// TIA Portal V15.1 export
// export: Created 2026-01-15T16:29:47.7440126Z, ExportSetting WithDefaults, WithReadOnly, DisplayName Totally Integrated Automation Portal, DisplayVersion V15.1 Update 8, DisplayName TIA Portal Openness, DisplayVersion V15.1 Update 8, DisplayName STEP 7 Professional, DisplayVersion V15.1 Update 8, DisplayName WinCC Advanced, DisplayVersion V15.1 Update 8
FUNCTION "FCXL_CCD_FD1" : Void   // FC10, LAD
{ S7_Optimized_Access := 'TRUE' }
VERSION : 0.1
// stored: AutoNumber true, CodeModifiedDate 2026-01-15T16:25:54.9008625Z, CompileDate 2026-01-15T16:25:54.9411388Z, CreationDate 2026-01-15T16:24:02.4619467Z, HandleErrorsWithinBlock false, InterfaceModifiedDate 2024-08-08T03:13:40.4539851Z, IsConsistent true, IsIECCheckEnabled false, IsKnowHowProtected false, IsWriteProtected false, LibraryConformanceStatus Error: The block contains calls of single instances. Warning: The object contains access to global data blocks. Warning: The block contains direct access to inputs, outputs, bit memories, indirect access to the registry or indirect access to external memory areas that are unknown at the time of compilation., ModifiedDate 2026-01-15T16:25:54.9008625Z, ParameterModified 2024-08-08T03:13:40.4539851Z, PLCSimAdvancedSupport false, SetENOAutomatically False, StructureModified 2024-08-08T03:13:40.4539851Z, UDAEnableTagReadback false
   VAR_TEMP   // added for the SCL form of the ladder/FBD networks
      _w1 : Bool;
      _w2 : Bool;
      _w3 : Bool;
   END_VAR
BEGIN

REGION Network 1: Cân CE/FD1 Full
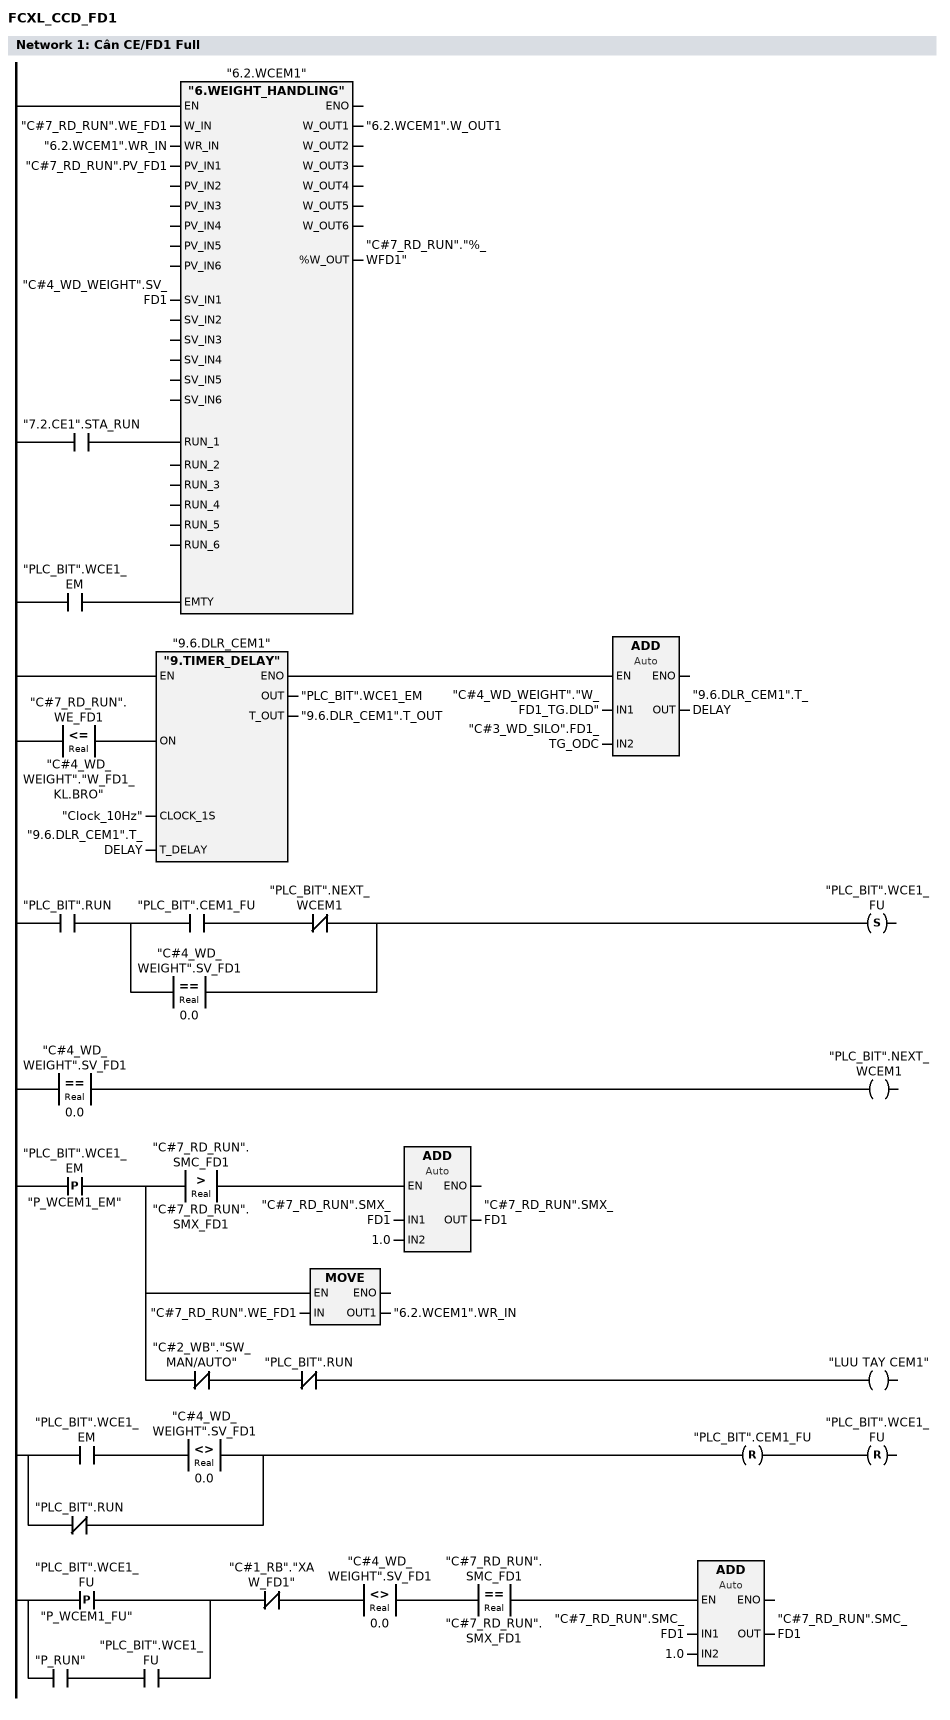
   RUNG wire#powerrail
      "6.2.WCEM1"(RUN_1 := wire#w1, EMTY := wire#w2, W_IN := "C#7_RD_RUN".WE_FD1, WR_IN := "6.2.WCEM1".WR_IN, PV_IN1 := "C#7_RD_RUN".PV_FD1, PV_IN2 :=, PV_IN3 :=, PV_IN4 :=, PV_IN5 :=, PV_IN6 :=, SV_IN1 := "C#4_WD_WEIGHT".SV_FD1, SV_IN2 :=, SV_IN3 :=, SV_IN4 :=, SV_IN5 :=, SV_IN6 :=, RUN_2 :=, RUN_3 :=, RUN_4 :=, RUN_5 :=, RUN_6 :=, W_OUT1 => "6.2.WCEM1".W_OUT1, W_OUT2 =>, W_OUT3 =>, W_OUT4 =>, W_OUT5 =>, W_OUT6 =>, "%W_OUT" => "C#7_RD_RUN"."%_WFD1")
   END_RUNG
   RUNG wire#powerrail
      Contact( "7.2.CE1".STA_RUN )
   END_RUNG wire#w1
   RUNG wire#powerrail
      Contact( "PLC_BIT".WCE1_EM )
   END_RUNG wire#w2
   RUNG wire#powerrail
      "9.6.DLR_CEM1"(ON := wire#w3, CLOCK_1S := "Clock_10Hz", T_DELAY := "9.6.DLR_CEM1".T_DELAY, OUT => "PLC_BIT".WCE1_EM, T_OUT => "9.6.DLR_CEM1".T_OUT)
      Add(in1 := "C#4_WD_WEIGHT"."W_FD1_TG.DLD", in2 := "C#3_WD_SILO".FD1_TG_ODC, out => "9.6.DLR_CEM1".T_DELAY)
   END_RUNG
   RUNG wire#powerrail
      { S7_Templates := "SrcType := Real" } LE_Contact(in1 := "C#7_RD_RUN".WE_FD1, in2 := "C#4_WD_WEIGHT"."W_FD1_KL.BRO")
   END_RUNG wire#w3
   RUNG wire#powerrail
      Contact( "PLC_BIT".RUN )
      wire#w4
      Contact( "PLC_BIT".CEM1_FU )
      I_Contact( "PLC_BIT".NEXT_WCEM1 )
      wire#w5
      S_Coil( "PLC_BIT".WCE1_FU )
   END_RUNG
   RUNG wire#w4
      { S7_Templates := "SrcType := Real" } EQ_Contact(in1 := "C#4_WD_WEIGHT".SV_FD1, in2 := 0.0)
   END_RUNG wire#w5
   RUNG wire#powerrail
      { S7_Templates := "SrcType := Real" } EQ_Contact(in1 := "C#4_WD_WEIGHT".SV_FD1, in2 := 0.0)
      Coil( "PLC_BIT".NEXT_WCEM1 )
   END_RUNG
   RUNG wire#powerrail
      P_Contact(operand := "PLC_BIT".WCE1_EM, bit := "P_WCEM1_EM")
      wire#w6
      { S7_Templates := "SrcType := Real" } GT_Contact(in1 := "C#7_RD_RUN".SMC_FD1, in2 := "C#7_RD_RUN".SMX_FD1)
      Add(in1 := "C#7_RD_RUN".SMX_FD1, in2 := 1.0, out => "C#7_RD_RUN".SMX_FD1)
   END_RUNG
   RUNG wire#w6
      Move(in := "C#7_RD_RUN".WE_FD1, out1 => "6.2.WCEM1".WR_IN)
   END_RUNG
   RUNG wire#w6
      I_Contact( "C#2_WB"."SW_MAN/AUTO" )
      I_Contact( "PLC_BIT".RUN )
      Coil( "LUU TAY CEM1" )
   END_RUNG
   RUNG wire#powerrail
      Contact( "PLC_BIT".WCE1_EM )
      { S7_Templates := "SrcType := Real" } NE_Contact(in1 := "C#4_WD_WEIGHT".SV_FD1, in2 := 0.0)
      wire#w7
      R_Coil( "PLC_BIT".CEM1_FU )
      R_Coil( "PLC_BIT".WCE1_FU )
   END_RUNG
   RUNG wire#powerrail
      I_Contact( "PLC_BIT".RUN )
   END_RUNG wire#w7
   RUNG wire#powerrail
      P_Contact(operand := "PLC_BIT".WCE1_FU, bit := "P_WCEM1_FU")
      wire#w8
      I_Contact( "C#1_RB"."XA W_FD1" )
      { S7_Templates := "SrcType := Real" } NE_Contact(in1 := "C#4_WD_WEIGHT".SV_FD1, in2 := 0.0)
      { S7_Templates := "SrcType := Real" } EQ_Contact(in1 := "C#7_RD_RUN".SMC_FD1, in2 := "C#7_RD_RUN".SMX_FD1)
      Add(in1 := "C#7_RD_RUN".SMC_FD1, in2 := 1.0, out => "C#7_RD_RUN".SMC_FD1)
   END_RUNG
   RUNG wire#powerrail
      Contact( "P_RUN" )
      Contact( "PLC_BIT".WCE1_FU )
   END_RUNG wire#w8
   // the same network as SCL:
   "6.2.WCEM1"(W_IN := "C#7_RD_RUN".WE_FD1,   // "6.WEIGHT_HANDLING"
               WR_IN := "6.2.WCEM1".WR_IN,
               PV_IN1 := "C#7_RD_RUN".PV_FD1,
               SV_IN1 := "C#4_WD_WEIGHT".SV_FD1,
               RUN_1 := "7.2.CE1".STA_RUN,
               EMTY := "PLC_BIT".WCE1_EM,
               W_OUT1 => "6.2.WCEM1".W_OUT1,
               "%W_OUT" => "C#7_RD_RUN"."%_WFD1");
   "9.6.DLR_CEM1"(ON := "C#7_RD_RUN".WE_FD1 <= "C#4_WD_WEIGHT"."W_FD1_KL.BRO",   // "9.TIMER_DELAY"
                  CLOCK_1S := "Clock_10Hz",
                  T_DELAY := "9.6.DLR_CEM1".T_DELAY,
                  OUT => "PLC_BIT".WCE1_EM,
                  T_OUT => "9.6.DLR_CEM1".T_OUT,
                  ENO => #_w1);
   IF #_w1 THEN "9.6.DLR_CEM1".T_DELAY := "C#4_WD_WEIGHT"."W_FD1_TG.DLD" + "C#3_WD_SILO".FD1_TG_ODC; END_IF;
   IF "PLC_BIT".RUN AND (("PLC_BIT".CEM1_FU AND NOT "PLC_BIT".NEXT_WCEM1) OR ("C#4_WD_WEIGHT".SV_FD1 = 0.0)) THEN
       "PLC_BIT".WCE1_FU := TRUE;
   END_IF;
   "PLC_BIT".NEXT_WCEM1 := "C#4_WD_WEIGHT".SV_FD1 = 0.0;
   #_w2 := "PLC_BIT".WCE1_EM AND NOT "P_WCEM1_EM";   // rising edge of "PLC_BIT".WCE1_EM
   "P_WCEM1_EM" := "PLC_BIT".WCE1_EM;
   IF #_w2 AND ("C#7_RD_RUN".SMC_FD1 > "C#7_RD_RUN".SMX_FD1) THEN
       "C#7_RD_RUN".SMX_FD1 := "C#7_RD_RUN".SMX_FD1 + 1.0;
   END_IF;
   IF #_w2 THEN "6.2.WCEM1".WR_IN := "C#7_RD_RUN".WE_FD1; END_IF;
   "LUU TAY CEM1" := #_w2 AND NOT "C#2_WB"."SW_MAN/AUTO" AND NOT "PLC_BIT".RUN;
   IF ("PLC_BIT".WCE1_EM AND ("C#4_WD_WEIGHT".SV_FD1 <> 0.0)) OR NOT "PLC_BIT".RUN THEN
       "PLC_BIT".CEM1_FU := FALSE;
       "PLC_BIT".WCE1_FU := FALSE;
   END_IF;
   #_w3 := "PLC_BIT".WCE1_FU AND NOT "P_WCEM1_FU";   // rising edge of "PLC_BIT".WCE1_FU
   "P_WCEM1_FU" := "PLC_BIT".WCE1_FU;
   IF (#_w3 OR ("P_RUN" AND "PLC_BIT".WCE1_FU)) AND NOT "C#1_RB"."XA W_FD1" AND ("C#4_WD_WEIGHT".SV_FD1 <> 0.0) AND ("C#7_RD_RUN".SMC_FD1 = "C#7_RD_RUN".SMX_FD1) THEN
       "C#7_RD_RUN".SMC_FD1 := "C#7_RD_RUN".SMC_FD1 + 1.0;
   END_IF;
END_REGION
END_FUNCTION
